{attribute addProperty BoxType "EK1100-0000-0018"}
{attribute addProperty Id "Beckhoff_ER6xxxEK1122Beckhoff_ER6xxxEK1122_7ED5D8733498437.25"}
{attribute addProperty CRC "971981903"}
{attribute addProperty SizeInBites "3498"}
{attribute addProperty SizeInBytes "437.25"}
TYPE Beckhoff_ER6xxx_39EF444F EXTENDS EK1100_179A0949 :
STRUCT
	{attribute addProperty Name "Beckhoff_ER6xxxEK1122"}
	Beckhoff_ER6xxxEK1122 : Beckhoff_ER6xxxEK1122_7ED5D873;
END_STRUCT
END_TYPE

(* stored: Version 1.2.0.0, ProductVersion 3.1.4024.9
   DUT Beckhoff_ER6xxx_39EF444F: Id {fb6295a9-80eb-400f-b537-c73550b5e659} *)
